KUKA KRL program: WeldSeam01.src, WeldSeam01.dat

--- WeldSeam01.src ---
&ACCESS RVP
&REL 1
&COMMENT Butt weld seam program
DEF WeldSeam01()
  ;FOLD INI
    ;FOLD BASISTECH INI
      BAS(#INITMOV, 0)
    ;ENDFOLD
  ;ENDFOLD

  PTP HOME Vel=100% DEFAULT

  ;FOLD LIN P1 Vel=2m/s CPDAT1 Tool[1] Base[2]
    LIN P1 Vel=2m/s CPDAT1 Tool[1] Base[2]
  ;ENDFOLD

  ;FOLD ARCON
    $OUT[1] = TRUE
  ;ENDFOLD

  ;FOLD LIN P2 Vel=10mm/s CPDAT2 Tool[1] Base[2]
    LIN P2 Vel=10mm/s CPDAT2 Tool[1] Base[2]
  ;ENDFOLD

  ;FOLD ARCOFF
    $OUT[1] = FALSE
  ;ENDFOLD

  PTP HOME Vel=100% DEFAULT

END

--- WeldSeam01.dat ---
DEFDAT WeldSeam01
  ;FOLD EXTERNAL DECLARATIONS; %{PE}
  ;ENDFOLD

  DECL E6POS HOME={A1 0.0, A2 -90.0, A3 90.0, A4 0.0, A5 0.0, A6 0.0}
  DECL E6POS P1={X 500.0, Y 200.0, Z 300.0, A 0.0, B 90.0, C 0.0, S 2, T 10}
  DECL E6POS P2={X 500.0, Y 800.0, Z 300.0, A 0.0, B 90.0, C 0.0, S 2, T 10}

  DECL REAL weld_speed=10.0
  DECL INT weld_mode=1

ENDDAT
